// TIA Portal V21 export
TYPE "switchgearAlm"
   STRUCT
      falseFb : Bool;
      sgNotReadyToStart : Bool;
      badFb : Bool;
      badOut : Bool;
      sticking : Bool;
      noFb : Bool;
      stepErr : Bool;
   END_STRUCT;
END_TYPE
